// TIA Portal V19 export
DATA_BLOCK "Decoiler2"   // DB49
// stored: InstanceOfName Decoiler_FB, InstanceOfType FB
"Decoiler_FB"
   // VAR_INPUT
   //    AreaInterface : "AreaInterface";
   //    ZSI : "udt_ZoneSafetyInterface";
   //    DSI : Struct
   //       Feed : "udt_DeviceSafetyInterface";
   //       Jaws : "udt_DeviceSafetyInterface";
   //       Coupling : "udt_DeviceSafetyInterface";
   //       SnubberLift : "udt_DeviceSafetyInterface";
   //       SnubberRoll : "udt_DeviceSafetyInterface";
   //    END_STRUCT;
   //    Drive : "TAx_DriveInterface";
   //    HW_ID_TEL1 : HW_SUBMODULE;
   //    DataIn : Struct
   //       DiameterSensor : Int;
   //       LsPosizioneRazza : Bool;
   //       Feed : "SpeedMachine_DataIn";
   //       Jaws : "ValveMachine_DataIn";
   //       Coupling : "ValveMachine_DataIn";
   //       SnubberLift : "ValveMachine_DataIn";
   //       SnubberRoll : "ValveMachine_DataIn";
   //       Loop : Struct
   //          Connector : Bool;
   //          S_MinHigh : Bool;
   //          S_SpeedAsjust : Bool;
   //          S_MaxLow : Bool;
   //       END_STRUCT;
   //       PneumaticBrake : Struct
   //          PbOpenClose : Bool;
   //          PbPartialOpenClose : Bool;
   //       END_STRUCT;
   //    END_STRUCT;
   //    CIn : Struct
   //       Manager : "Decoiler_Manager";
   //       PressureRunning : Bool;
   //    END_STRUCT;
   //    Config : Struct
   //       Loop : Struct
   //          Exist_S_MinHigh : Bool;
   //          Exist_S_SpeedAdjust : Bool;
   //       END_STRUCT;
   //       Feed : "SpeedMachine_Config";
   //       Jaws : "ValveMachine_Config";
   //       Coupling : "ValveMachine_Config";
   //       SnubberLift : "ValveMachine_Config";
   //       SnubberRoll : "ValveMachine_Config";
   //       Enable_End_Of_Coil_Using_Loop : Bool;
   //    END_STRUCT;
   // END_VAR
   // VAR_OUTPUT
   //    MachineInterface : "MachineInterface";
   //    DataOut : Struct
   //       Feed : "SpeedMachine_DataOut";
   //       Jaws : "ValveMachine_DataOut";
   //       Coupling : "ValveMachine_DataOut";
   //       SnubberLift : "ValveMachine_DataOut";
   //       SnubberRoll : "ValveMachine_DataOut";
   //       PneumaticBrake : Struct
   //          V_Open : Bool;
   //          V_PartialHigh : Bool;
   //          V_PartialLow : Bool;
   //          Lp_PbPartialBrake : Bool;
   //       END_STRUCT;
   //    END_STRUCT;
   //    COut : "Decoiler_Status";
   // END_VAR
   // VAR_IN_OUT
   //    PersistentValues : "Decoiler_Pers";
   // END_VAR
   // VAR
   //    Alarm : Struct
   //       Feed : "SpeedMachine_Alr";
   //       Jaws : "ValveAlr";
   //       Coupling : "ValveAlr";
   //       SnubberLift : "ValveAlr";
   //       SnubberRoll : "ValveAlr";
   //       DimeterSensor : Struct
   //          SensorrPresetNeed { ExternalAccessible := 'False'; ExternalVisible := 'False'; ExternalWritable := 'False'} : Bool;
   //       END_STRUCT;
   //       Loop : Struct
   //          ConnectorUnplugged : Bool;
   //       END_STRUCT;
   //    END_STRUCT;
   //    Warning : Struct
   //       EndCoilDetect : Bool;
   //       Feed : "SpeedMachine_Wng";
   //       Jaws : "ValveMachine_Wng";
   //       Coupling { S7_SetPoint := 'True'} : "ValveMachine_Wng";
   //       SnubberLift { S7_SetPoint := 'True'} : "ValveMachine_Wng";
   //       SnubberRoll { S7_SetPoint := 'True'} : "ValveMachine_Wng";
   //       Loop : Struct
   //          MinHigh : Bool;
   //       END_STRUCT;
   //    END_STRUCT;
   //    HMI : Struct
   //       Diameter_ButtonPreset : Bool;
   //       Diameter_PresetValue : Real;
   //    END_STRUCT;
   //    Sts : Struct
   //       StopPosizioneRazza : Bool;
   //    END_STRUCT;
   //    Ctrl : Struct
   //       Jaws : Struct
   //          AutoOpen : Bool;
   //          TON_Pause : IEC_TIMER;
   //          TON_Duration : IEC_TIMER;
   //       END_STRUCT;
   //       Brake : Struct
   //          Open_ReqByMotor : Bool;
   //          TON_PartialOFF : IEC_TIMER;
   //          TON_OpenOFF : IEC_TIMER;
   //       END_STRUCT;
   //    END_STRUCT;
   //    DiameterSensor { S7_SetPoint := 'True'} : "Decoiler_DiameterSensor_FB";
   //    Loop { S7_SetPoint := 'True'} : "Decoiler_Loop_FB";
   //    Feed { S7_SetPoint := 'True'} : "SpeedMachine_FB";
   //    PneumaticBrake { S7_SetPoint := 'True'} : "Decoiler_PneumaticBrake";
   //    Jaws { S7_SetPoint := 'True'} : "ValveMachine_FB";
   //    SnubberLift { S7_SetPoint := 'True'} : "ValveMachine_FB";
   //    SnubberRoll { S7_SetPoint := 'True'} : "ValveMachine_FB";
   //    Coupling { S7_SetPoint := 'True'} : "ValveMachine_FB";
   //    TON_EndCoilDetect : IEC_TIMER;
   //    AuxPE : Struct
   //       LsPosizioneRazza : Bool;
   //    END_STRUCT;
   // END_VAR
BEGIN
END_DATA_BLOCK
